# EPICS autosave request: ADVimba/iocs/vimbaIOC/iocBoot/iocVimba/auto_settings.req
file "vimba_settings.req",                P=$(P),  R=cam1:
file "NDStdArrays_settings.req",          P=$(P),  R=image1:
file "commonPlugin_settings.req",         P=$(P)
